FUNCTION FUN_Scale : REAL
VAR_INPUT
	ix :UINT;
	ix_max :REAL;
	ix_min :REAL;
	ry_min :REAL;
	ry_max :REAL;
END_VAR
VAR
	rk :REAL :=0.0854492188; //für Dispenser Ultraschallsensor 
	rd :REAL :=0;
END_VAR

//FUN keine deklarierung im Hauptprogramm

rk:=(ry_max-ry_min)/(ix_max-ix_min);
rd:=ry_min-rk*ix_min;

FUN_Scale := rk*ix+rd;

IF FUN_Scale > ry_max THEN
	FUN_Scale:=ry_max;
ELSIF FUN_Scale < ry_min THEN
	FUN_Scale:=ry_min;
END_IF

END_FUNCTION

(* stored: Version 1.1.0.1, ProductVersion 3.1.4024.15
   POU FUN_Scale: Id {44f48920-fa01-4344-bf7b-5c55ad611afa}, SpecialFunc None *)
